FUNCTION Convert_TOD_TO_WORD : BOOL
VAR_INPUT
	in : TOD;
	out : REFERENCE TO WORD;
END_VAR
VAR
	converted : WORD;
END_VAR

converted := TOD_TO_WORD(in);

IF (WORD_TO_TOD(converted) <> in) THEN
	RETURN;
END_IF

out := converted;
Convert_TOD_TO_WORD := TRUE;

END_FUNCTION

(* stored: Version 1.1.0.1, ProductVersion 3.1.4024.12
   POU Convert_TOD_TO_WORD: Id {e5cf9853-f56b-4e74-a13e-2464172cdf99}, SpecialFunc None *)
